TYPE typ_MotionGearing :
STRUCT
	MC_GearIn					: MC_GearIn;
	MC_GearInDyn				: MC_GearInDyn;
	MC_GearInMultiMaster		: MC_GearInMultiMaster;
	MC_GearOut					: MC_GearOut;
END_STRUCT
END_TYPE

(* stored: Version 1.1.0.1, ProductVersion 3.1.4022.17
   DUT typ_MotionGearing: Id {158c8988-5041-4a0d-a7d1-0693b1935a89} *)
